// TIA Portal V17 export
// export: Created 2022-10-06T11:58:03.6054276Z, ExportSetting WithDefaults, DisplayName Totally Integrated Automation Portal, DisplayVersion V17, DisplayName TIA Portal Openness, DisplayVersion V17, DisplayName TIA Portal Version Control Interface, DisplayVersion V17, DisplayName SINAMICS Startdrive Advanced, DisplayVersion V17, DisplayName SINAMICS Startdrive G130, G150, S120, S150, SINAMICS MV, S210, DisplayVersion V17, DisplayName SINAMICS Startdrive G110M, G120, G120C, G120D, G120P, G115D, DisplayVersion V17, DisplayName STEP 7 Professional, DisplayVersion V17, DisplayName STEP 7 Safety, DisplayVersion V17, DisplayName WinCC Advanced, DisplayVersion V17
VAR_GLOBAL   // PLC tag table "Default tag table"
   "jaw latch" AT %M0.0 : Bool;
   "jaw output" AT %M0.1 : Bool;
   "prog reset" AT %M0.2 : Bool;
   TempVar AT %MW2 : Word;
   AlwaysOn AT %M0.3 : Bool;
   StartLatch AT %M0.4 : Bool;
   StartLatchBit AT %M0.5 : Bool;
END_VAR
